{attribute addProperty BoxType "AT2041-0250-0023"}
{attribute addProperty Id "A_0099_AT2040_5250_0018_AT2040_5250AT2040_C5E5984862678.25"}
{attribute addProperty CRC "1551186803"}
{attribute addProperty SizeInBites "626"}
{attribute addProperty SizeInBytes "78.25"}
TYPE A_0045_AT2041_0250_0023_5C753B73 EXTENDS AT2041_BA5A9548 :
STRUCT
	{attribute addProperty Name "A_0099_AT2040_5250_0018_AT2040_5250"}
	A_0099_AT2040_5250_0018_AT2040_5250 : AT2040_C5E59848;
END_STRUCT
END_TYPE

(* stored: Version 1.2.0.0, ProductVersion 3.1.4024.9
   DUT A_0045_AT2041_0250_0023_5C753B73: Id {87323569-7151-49d5-8bbe-5414b766fe82} *)
